{attribute 'GeneratedUsingTerminal: EL2521-0124-0016'}
{attribute addProperty BoxType "EL2521-0124-0016"}
{attribute addProperty Id "PTO_StatusAT %I*PTO_Status_C6D3EC315ENC_Status_compactAT %I*ENC_Status_compact_64F890EB11PLS_StatusAT %I*PLS_Status_A60F49334PTO_ControlAT %Q*PTO_Control_392B4D2E5ENC_Control_compactAT %Q*ENC_Control_compact_DC4E290B5PLS_Control_compactAT %Q*PLS_Control_compact_DC91A7B86WcStateAT %I*WcState_9091E0EB2InfoDataAT %I*InfoData_94A18F5E2"}
{attribute addProperty CRC "1670877012"}
{attribute addProperty Size "40"}
TYPE EL2521_63978F54 EXTENDS EtcSlaveTerminalBase_947E5A46 :
STRUCT
	{attribute addProperty Name "PTO_Status"}
	PTO_Status : PTO_Status_C6D3EC31;
	{attribute addProperty Name "ENC_Status_compact"}
	ENC_Status_compact : ENC_Status_compact_64F890EB;
	{attribute addProperty Name "PLS_Status"}
	PLS_Status : PLS_Status_A60F4933;
	{attribute addProperty Name "PTO_Control"}
	PTO_Control : PTO_Control_392B4D2E;
	{attribute addProperty Name "ENC_Control_compact"}
	ENC_Control_compact : ENC_Control_compact_DC4E290B;
	{attribute addProperty Name "PLS_Control_compact"}
	PLS_Control_compact : PLS_Control_compact_DC91A7B8;
	{attribute addProperty Name "WcState"}
	WcState : WcState_9091E0EB;
	{attribute addProperty Name "InfoData"}
	InfoData : InfoData_94A18F5E;
END_STRUCT
END_TYPE

(* stored: Version 1.2.0.0, ProductVersion 3.1.4024.9
   DUT EL2521_63978F54: Id {2e7f4d4c-b5d2-4be6-a0f1-25f7c49b3ea1} *)
